{attribute 'qualified_only'}
{attribute 'strict'}
TYPE eNetcontMode :
(
	auto := 0,
	left := 1,
	right := 2,
	none := 3
);
END_TYPE

(* stored: Version 1.1.0.1, ProductVersion 3.1.4026.18
   DUT eNetcontMode: Id {6466fd48-f991-44c1-a93d-72587edb025b} *)
